{attribute addProperty BoxType "AT2041-0250-0018"}
{attribute addProperty Id "A_0104_AT2042_5250_0019_AT2042_5250AT2042_C5E5984862678.25"}
{attribute addProperty CRC "1502877408"}
{attribute addProperty SizeInBites "626"}
{attribute addProperty SizeInBytes "78.25"}
TYPE A_0040_AT2041_0250_0018_599416E0 EXTENDS AT2041_BA5A9548 :
STRUCT
	{attribute addProperty Name "A_0104_AT2042_5250_0019_AT2042_5250"}
	A_0104_AT2042_5250_0019_AT2042_5250 : AT2042_C5E59848;
END_STRUCT
END_TYPE

(* stored: Version 1.2.0.0, ProductVersion 3.1.4024.9
   DUT A_0040_AT2041_0250_0018_599416E0: Id {06820555-546c-4021-ac40-f535398f2cc9} *)
